{attribute 'linkalways'} 
{attribute 'no_explicit_call' := 'This FB is a CLASS and must be accessed using methods or properties'}
{attribute 'enable_dynamic_creation'}
FUNCTION_BLOCK FINAL XOR_UDINT EXTENDS Node
VAR
	in1 : _UDINT(0);
	in2 : _UDINT(0);
	out : _UDINT(0);
END_VAR

METHOD PUBLIC Clone : I_Node
VAR
	pNode : POINTER TO XOR_UDINT;
END_VAR
pNode := __NEW(XOR_UDINT);
Clone := pNode^;
END_METHOD

METHOD FB_init : BOOL
VAR_INPUT
	bInitRetains : BOOL; // if TRUE, the retain variables are initialized (warm start / cold start)
	bInCopyCode : BOOL;  // if TRUE, the instance afterwards gets moved into the copy code (online change)
END_VAR
AddInput('in1',THIS^.in1);
AddInput('in2',THIS^.in2);
AddOutput('out', THIS^.out);
END_METHOD

METHOD PROTECTED OnExecute
VAR
END_VAR
out.Value := in1.Value XOR in2.Value;
END_METHOD

END_FUNCTION_BLOCK

(* stored: Version 1.1.0.1, ProductVersion 3.1.4024.15
   POU XOR_UDINT: Id {f1b976dd-1e1f-4954-bf97-7c3b0dd9a79d}, SpecialFunc None
   Folder Constructor: Id {d313a471-bb5f-4e9a-9ac3-d7ef0d062978}
   Method Clone: Id {fc885844-4a7a-40cb-87b3-9ab05df36aa7}
   Method FB_init: Id {28d26c7b-e6ad-4d41-8f87-91643f662208}
   Method OnExecute: Id {35659347-8b0d-4fbd-8e4d-de71f819c88c} *)
